{attribute 'qualified_only'}
VAR_GLOBAL CONSTANT
END_VAR

(* stored: Version 1.1.0.1, ProductVersion 3.1.4024.10
   GVL GVL: Id {e5c78160-cbbb-43f9-8e79-03ff05bb6daf}, ParameterList True *)
